Yaskawa INFORM job: POS_TEST2.JBI

/JOB
//NAME POS_TEST2
//POS
///NPOS 2,0,0,0,0,0
///TOOL 0
///POSTYPE BASE
///RECTAN
C00000=1975.000,-715.000,-849.000,-180.0000,0.0000,0.0000
C00001=1975.000,785.000,-849.000,-180.0000,0.0000,0.0000
//INST
///DATE 2023/01/30 14:00
///ATTR SC,RW,RJ
////FRAME BASE
///GROUP1 RB1
NOP
MOVJ C00000 VJ=0.78
MOVL C00001 V=100.0
END
